// Brief: Master Arm Error Hold
FUNCTION_BLOCK PUBLIC FB_StateCtrlError EXTENDS FB_MasterArmCtrlBase
VAR_INPUT
END_VAR
VAR_OUTPUT
END_VAR
VAR
END_VAR

METHOD PUBLIC init : BOOL
VAR_IN_OUT CONSTANT
	i_masterArm	:FB_MasterArm;
END_VAR
VAR_IN_OUT 
	r_masterArmCtrlCmd :ST_ArmCtrlCmds;
END_VAR

VAR
	i:INT;
END_VAR
SUPER^.Init(i_masterArm,r_masterArmCtrlCmd);

//disable joints which is error
FOR i := 1 TO g_mJntNum DO
	IF SafetyCheck.m_SafetyCheck.m_jntErrFlag[i_masterArm.armIdx, i, 2] OR SafetyCheck.m_SafetyCheck.m_jntErrFlag[i_masterArm.armIdx, i, 3] THEN
		m_jntEnableFlag[i] := 0;
	ELSE
		m_jntEnableFlag[i] := 1;
	END_IF
END_FOR

// update commands to arm
copyCmds(r_masterArmCtrlCmd);
END_METHOD

END_FUNCTION_BLOCK

(* stored: Version 1.1.0.1, ProductVersion 3.1.4024.12
   POU FB_StateCtrlError: Id {78b2e60d-537e-446e-8b3b-6db63d5ab02c}, SpecialFunc None
   Method init: Id {e6a6f329-eae4-4e64-b8ba-0dd027b37a8e} *)
